// TIA Portal V18 export
DATA_BLOCK "FC1521_EnviroPro_TCPClient_DB"   // DB4
VERSION : 0.1
// stored: AutoNumber true, DBAccessibleFromOPCUA true, DBAccessibleFromWebserver true, InstanceOfName FB1521_EnviroPro_TCPClient, InstanceOfType FB
"FB1521_EnviroPro_TCPClient"
   // VAR_INPUT
   //    Enable : Bool;
   //    EN_R : Bool;
   //    ID : CONN_OUC;
   //    PORT : UInt;
   //    IP_1 : Byte;
   //    IP_2 : Byte;
   //    IP_3 : Byte;
   //    IP_4 : Byte;
   // END_VAR
   // VAR_OUTPUT
   //    RCV_DONE : Bool;
   //    RCV_BUSY : Bool;
   //    RCV_ERROR : Bool;
   //    RCV_STATUS : Word;
   //    SEND_DONE : Bool;
   //    SEND_BUSY : Bool;
   //    SEND_ERROR : Bool;
   //    SEND_STATUS : Word;
   // END_VAR
   // VAR_IN_OUT
   //    COM_RST : Bool;
   // END_VAR
   // VAR
   //    CONNECT : TCON_IP_v4;
   //    RCV_DATA : Array[1..90] of Char;
   //    RCV_VWC : Array[1..9] of Real;
   //    RCV_ECe : Array[1..9] of Real;
   //    RCV_TEMP : Array[1..9] of Real;
   //    Done_Old : Bool;
   //    Pos_R : Int;
   //    TRCV_C : TRCV_C;
   //    TSEND_C { S7_SetPoint := 'True'} : TSEND_C;
   //    Send_Cmd : String[12];
   //    Count_Cmd : Int;
   //    TON_1 { S7_SetPoint := 'True'} : TON_TIME;
   //    TON_2 { S7_SetPoint := 'True'} : TON_TIME;
   //    QT1 { ExternalAccessible := 'False'; ExternalVisible := 'False'; ExternalWritable := 'False'} : Bool;
   //    QT2 { ExternalAccessible := 'False'; ExternalVisible := 'False'; ExternalWritable := 'False'} : Bool;
   // END_VAR
BEGIN
END_DATA_BLOCK
